(* PLC project Tc3_MC2_AdvancedHoming.MC_StepBlock Demo, tc3-libraries-kb TwinCAT 3.1 *)
(* stored: creationDateTime 2026-05-25T00:00:00, modificationDateTime 2026-05-25T00:00:00 *)

PROGRAM P_Demo_MC_StepBlock
  VAR
    fbStepBlock : MC_StepBlock;
    axisHoming : AXIS_REF;  (* 归零目标轴；运行前需先 MC_Power 使能 *)
    rtExec : R_TRIG;  (* 把保持型请求位整成单次上升沿 *)
    bBlockReq : BOOL := FALSE;  (* 在线置 TRUE 触发一次执行 *)
    homingParam : MC_HomingParameter;  (* 贯穿整条归零序列、各 FB 间逐级传递的参数结构 *)
    homingOptions : ST_Home_Options3;  (* 选项结构，Beckhoff 伺服保持默认（DisableDriveAccess := FALSE） *)
    bBlockDone : BOOL;
    bBusy : BOOL;
    bBlockActive : BOOL;
    bAborted : BOOL;
    bError : BOOL;
    nErrorID : UDINT;
  END_VAR

// 场景：无开关无零脉冲的推料电动轴，用低速撞机械硬止挡来定零。限矩 30% 防撞坏，
//       转矩达限且速度持续低于阈值即判定顶到止挡，把该点定为坐标 0。
// 价值：省去开关接线与调试，靠转矩+速度双判据可靠判断顶到止挡。
// 验证：先 MC_Power 使能；在线写 bBlockReq := TRUE，观察 bBlockActive TRUE，轴低速朝正向
//       顶；顶到止挡转矩升到限值、速度跌到 1 以下持续 200ms 后 bBlockDone TRUE，位置读数变 0。

// 把保持型在线请求位整成单次上升沿，避免持续触发（charter: Execute 用 R_TRIG）
rtExec(CLK := bBlockReq);

// 单次完整调用：所有 VAR_INPUT 显式赋值，Axis（及 Parameter）按 VAR_IN_OUT 必须传引用
fbStepBlock(
    Execute                := rtExec.Q,
    Direction              := mcPositiveDirection,
    Velocity               := 10.0,
    Acceleration           := 0.0,
    Deceleration           := 0.0,
    Jerk                   := 0.0,
    SetPosition            := 0.0,
    DetectionVelocityLimit := 1.0,
    DetectionVelocityTime  := T#200MS,
    TimeLimit              := T#20S,
    DistanceLimit          := 500.0,
    TorqueLimit            := 30.0,
    TorqueTolerance        := 5.0,
    BufferMode             := MC_Aborting,
    Options                := homingOptions,
    Done                   => bBlockDone,
    Busy                   => bBusy,
    Active                 => bBlockActive,
    CommandAborted         => bAborted,
    Error                  => bError,
    ErrorID                => nErrorID,
    Axis                   := axisHoming,
    Parameter              := homingParam);

// stateful 输出复位：请求复位后清掉本地观察位，便于下次干净触发
IF NOT bBlockReq AND NOT bBusy THEN
    bBlockDone := FALSE;
    bAborted := FALSE;
END_IF;
END_PROGRAM
